// TIA Portal project "MB_SERVER_TCP_1200" (V17)

(* hardware
DEVICE "S7-1200 station_1"  S7-1200 Station
   slot 0: "Rack_0"  S7-1200 Rack  Rack  V1.0
   slot 1: "PLC_1"  CPU 1211C DC/DC/DC  6ES7 211-1AE40-0XB0  V4.5
*)

// ===== PLC "PLC_1"  CPU 1211C DC/DC/DC =====

VAR_GLOBAL   // PLC tag table "Default tag table"
   "System_Byte" AT %MB1 : Byte;
   "FirstScan" AT %M1.0 : Bool;
   "DiagStatusUpdate" AT %M1.1 : Bool;
   "AlwaysTRUE" AT %M1.2 : Bool;
   "AlwaysFALSE" AT %M1.3 : Bool;
   "Clock_Byte" AT %MB0 : Byte;
   "Clock_10Hz" AT %M0.0 : Bool;
   "Clock_5Hz" AT %M0.1 : Bool;
   "Clock_2.5Hz" AT %M0.2 : Bool;
   "Clock_2Hz" AT %M0.3 : Bool;
   "Clock_1.25Hz" AT %M0.4 : Bool;
   "Clock_1Hz" AT %M0.5 : Bool;
   "Clock_0.625Hz" AT %M0.6 : Bool;
   "Clock_0.5Hz" AT %M0.7 : Bool;
END_VAR

DATA_BLOCK "MB-DB"   // DB2
{ S7_Optimized_Access := 'TRUE' }
VERSION : 0.1
   VAR
      CONNECT : TCON_IP_v4;
      DISCONNECT : Bool;
      NDR : Bool;
      DR : Bool;
      ERROR : Bool;
      STATUS : Word;
   END_VAR
BEGIN
   CONNECT.InterfaceId := 64;
   CONNECT.ID := 1;
   CONNECT.ConnectionType := 11;
   CONNECT.ActiveEstablished := false;
   CONNECT.RemoteAddress.ADDR[1] := 192;
   CONNECT.RemoteAddress.ADDR[2] := 168;
   CONNECT.RemoteAddress.ADDR[3] := 2;
   CONNECT.RemoteAddress.ADDR[4] := 153;
   CONNECT.RemotePort := 0;
   CONNECT.LocalPort := 502;
END_DATA_BLOCK

DATA_BLOCK "MB_HOLD_REG"   // DB3
{ S7_Optimized_Access := 'TRUE' }
VERSION : 0.1
   VAR
      "HOLD-REG" : Array[0..49] of Int;
   END_VAR
BEGIN
END_DATA_BLOCK

FUNCTION "MB-SERVER" : Void   // FC1, LAD
{ S7_Optimized_Access := 'TRUE' }
VERSION : 0.1
BEGIN

REGION Network 1
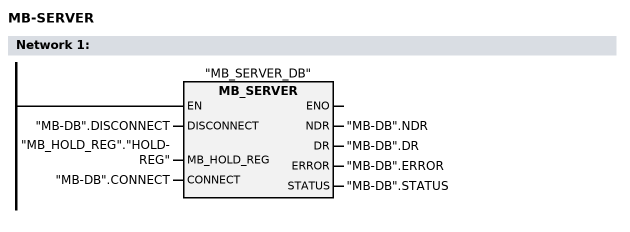
   "MB_SERVER_DB"(DISCONNECT := "MB-DB".DISCONNECT,   // MB_SERVER
                  MB_HOLD_REG := "MB_HOLD_REG"."HOLD-REG",
                  CONNECT := "MB-DB".CONNECT,
                  NDR => "MB-DB".NDR,
                  DR => "MB-DB".DR,
                  ERROR => "MB-DB".ERROR,
                  STATUS => "MB-DB".STATUS);
END_REGION
END_FUNCTION

ORGANIZATION_BLOCK "Main"   // OB1, LAD, ProgramCycle
TITLE = "Main Program Sweep (Cycle)"
{ S7_Optimized_Access := 'TRUE' }
VERSION : 0.1
   VAR_INPUT
      Initial_Call : Bool;   // Initial call of this OB
      Remanence : Bool;   // =True, if remanent data are available
   END_VAR
BEGIN

REGION Network 1
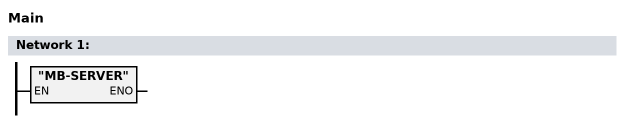
   RUNG wire#powerrail
      "MB-SERVER"()
   END_RUNG
   // the same network as SCL:
   "MB-SERVER"();
END_REGION
END_ORGANIZATION_BLOCK